(* IEC 61131-3 sources: Std_PalletMover/Class/I_LedControl, 1 file *)

(* ---- I_LedControl.st ---- *)
(*!
<Class
	Name               = "I_LedControl"
	Revision           = "0.0"
	RealtimeTask       = "false"
	CyclicTask         = "false"
	BackgroundTask     = "false"
	Sigmatek           = "false"
	OSInterface        = "false"
	HighPriority       = "false"
	Automatic          = "false"
	UpdateMode         = "Prescan"
	SharedCommandTable = "true"
	Objectsize         = "(570,120)">
	<Channels>
		<Server Name="ClassSvr" Visualized="false" Initialize="false" WriteProtected="true" Retentive="false"/>
		<Server Name="SetLeds" Visualized="false" Initialize="false" WriteProtected="true" Retentive="false"/>
	</Channels>
</Class>
*)
I_LedControl : CLASS
	TYPE
	  LedBinking :
	  (
	    LedAlwaysOn,
	    LedBlinking
	  )$UDINT;
	  LedState :  //! <Type Public="true" Name="LedState"/>
	  (
	    LedAllOff,
	    LedRed,
	    LedRedLeft,
	    LedRedRight,
	    LedGreen,
	    LedGreenLeft,
	    LedGreenRight,
	    LedBlue,
	    LedBlueLeft,
	    LedBlueRight
	  )$UDINT;
	END_TYPE
  //Servers:
	ClassSvr 	: SvrChCmd_DINT;
	SetLeds 	: SvrCh_LedState_PTofCls_I_LedControl;
  //Clients:
  //Variables:
  //Functions:
  //Tables:
	FUNCTION @STD
		VAR_OUTPUT
			ret_code	: CONFSTATES;
		END_VAR;
	FUNCTION GLOBAL TAB @CT_;
END_CLASS;
